FUNCTION_BLOCK DM_KRNL (* Device Management Kernel Block *)
  (* Standard: 61499 Demo ITA *)
  (* Version 0.3, 2001-01-22, JHC, Rockwell Automation, Corrected initialization, interfaced to FBManager *)
  (* Version 0.2, 2000-07-24, JHC, Rockwell Automation, Modified to use new DEV_MGR. *)
  (* Version 0.1, 2000-05-16, JHC, Rockwell Automation, File type changed to ".fbt" *)
  (* Version 0.0, 2000-03-18, JHC, Rockwell Automation *)
  (* Compiler header: package fb.rt; import fb.rt.net.*; *)
  (* Compiler Java IBM VisualAge 3.0 *)
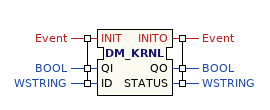
  EVENT_INPUT
    INIT WITH QI, ID; (* Service Initialization/Termination *)
  END_EVENT
  EVENT_OUTPUT
    INITO WITH QO, STATUS; (* Initialization/Termination Confirm *)
  END_EVENT
  VAR_INPUT
    QI : BOOL; (* 1=Initiate,0=Terminate *)
    ID : WSTRING; (* Server ID *)
  END_VAR
  VAR_OUTPUT
    QO : BOOL; (* 1=Initiated,0=Terminated *)
    STATUS : WSTRING; (* "OK"or Reason for Termination *)
  END_VAR
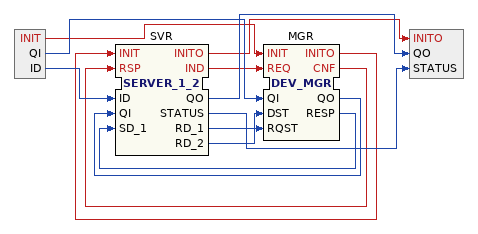
  FBS
    SVR : SERVER_1_2;
    MGR : DEV_MGR;
  END_FBS
  EVENT_CONNECTIONS
    INIT TO MGR.INIT;
    MGR.INITO TO SVR.INIT;
    SVR.INITO TO INITO;
    SVR.IND TO MGR.REQ;
    MGR.CNF TO SVR.RSP;
  END_CONNECTIONS
  DATA_CONNECTIONS
    QI TO MGR.QI;
    ID TO SVR.ID;
    MGR.QO TO SVR.QI;
    SVR.QO TO QO;
    SVR.STATUS TO STATUS;
    SVR.RD_1 TO MGR.DST;
    SVR.RD_2 TO MGR.RQST;
    MGR.RESP TO SVR.SD_1;
  END_CONNECTIONS
END_FUNCTION_BLOCK
